Staubli VAL3: Simas.dtx

mdesc mNomSpeed
frame fFrame1 = {x=0.000, y=0.000, z=0.000, rx=-0.000, ry=0.000, rz=-0.000, fatherId=world[0]}
dio Input[16]
  [0] = {link=BasicIO-2\%I0}
  [1] = {link=BasicIO-2\%I1}
  [2] = {link=BasicIO-2\%I2}
  [3] = {link=BasicIO-2\%I3}
  [4] = {link=BasicIO-2\%I4}
  [5] = {link=BasicIO-2\%I5}
  [6] = {link=BasicIO-2\%I6}
  [7] = {link=BasicIO-2\%I7}
  [8] = {link=BasicIO-2\%I8}
  [9] = {link=BasicIO-2\%I9}
  [10] = {link=BasicIO-2\%I10}
  [11] = {link=BasicIO-2\%I11}
  [12] = {link=BasicIO-2\%I12}
  [13] = {link=BasicIO-2\%I13}
  [14] = {link=BasicIO-2\%I14}
  [15] = {link=BasicIO-2\%I15}
dio Output[16]
  [0] = {link=BasicIO-2\%Q0}
  [1] = {link=BasicIO-2\%Q1}
  [2] = {link=BasicIO-2\%Q2}
  [3] = {link=BasicIO-2\%Q3}
  [4] = {link=BasicIO-2\%Q4}
  [5] = {link=BasicIO-2\%Q5}
  [6] = {link=BasicIO-2\%Q6}
  [7] = {link=BasicIO-2\%Q7}
  [8] = {link=BasicIO-2\%Q8}
  [9] = {link=BasicIO-2\%Q9}
  [10] = {link=BasicIO-2\%Q10}
  [11] = {link=BasicIO-2\%Q11}
  [12] = {link=BasicIO-2\%Q12}
  [13] = {link=BasicIO-2\%Q13}
  [14] = {link=BasicIO-2\%Q14}
  [15] = {link=BasicIO-2\%Q15}
tool tCurrentTool = {x=0.000, y=0.000, z=0.000, rx=-0.000, ry=0.000, rz=-0.000, fatherId=flange[0], ioLink=valve1}
mdesc mCurrentSpeed
pointRx pPointRx = {fatherId=fFrame1[0]}
pointRx pPointRx2 = {fatherId=fFrame1[0]}
